PROGRAM RTC 
VAR
	FB_LocalSystemTime_0	: FB_LocalSystemTime;
	TimeStamp		: TIMESTRUCT;
		
	TimeStamp_GMT		: TIMESTRUCT;
	
	FB_GetTimeZoneInformation_0 :FB_GetTimeZoneInformation;
	FB_SetTimeZoneInformation_0	:FB_SetTimeZoneInformation;
	ST_TimeZoneInformation:ST_TimeZoneInformation;

	
	Timer :ton;
	FlagGetTimeZone:BOOL;// :=TRUE;
	FlagSetTimeZone:BOOL;// :=TRUE;
	FlagInit	   :BOOL :=TRUE;	
	
	ErrorIDGetTimeZone:UDINT;
	ErrorIDSetTimeZone:UDINT;
	
	FB_TzSpecificLocalTimeToSystemTime:FB_TzSpecificLocalTimeToSystemTime;
//	amsid:T_AmsNetID :='192.168.101.2.1.1' ;
	amsid:T_AmsNetID ;
	
	//IISreset
	NT_StartProcess:NT_StartProcess;
	Flagiisreset:BOOL;
END_VAR

//Timer(IN:=FlagInit,PT:=T#5S,Q=>FlagGetTimeZone);

FB_LocalSystemTime_0(
	sNetID:= '' , 
	bEnable:= TRUE, 
	dwCycle:= , 
	dwOpt:= , 
	tTimeout:= , 
	bValid=> , 
	systemTime=> TimeStamp, 
	tzID=> );

IF FlagInit THEN
	FlagGetTimeZone:=TRUE;
	Flagiisreset:=TRUE;
	FlagInit:=FALSE;
	
END_IF	

	FB_GetTimeZoneInformation_0(bExecute := FlagGetTimeZone,sNetID:=PcTransmit.fbPcTransmit_0.RTC_amsid);
	IF FB_GetTimeZoneInformation_0.bError THEN
		FlagGetTimeZone:=FALSE;
		ErrorIDGetTimeZone:=FB_GetTimeZoneInformation_0.nErrID;
		FB_GetTimeZoneInformation_0(bExecute := FlagGetTimeZone);   		
	ELSIF FB_GetTimeZoneInformation_0.bBusy=FALSE AND FlagGetTimeZone THEN
		ST_TimeZoneInformation:=FB_GetTimeZoneInformation_0.tzInfo;	
		FlagGetTimeZone:=FALSE;
		FlagSetTimeZone:=TRUE;
		FB_GetTimeZoneInformation_0(bExecute := FlagGetTimeZone);	
	END_IF


	FB_SetTimeZoneInformation_0(bExecute:=FlagSetTimeZone, tzInfo:=ST_TimeZoneInformation);
	IF FB_SetTimeZoneInformation_0.bError THEN
		FlagSetTimeZone:=FALSE;
		ErrorIDSetTimeZone:=FB_SetTimeZoneInformation_0.nErrID;
		FB_SetTimeZoneInformation_0(bExecute := FlagSetTimeZone);   		
	ELSIF FB_SetTimeZoneInformation_0.bBusy=FALSE AND FlagSetTimeZone THEN
		FlagSetTimeZone:=FALSE;
		FB_SetTimeZoneInformation_0(bExecute := FlagGetTimeZone);	
	END_IF
	

FB_TzSpecificLocalTimeToSystemTime(in:=TimeStamp,tzInfo:=ST_TimeZoneInformation, out=>TimeStamp_GMT);

(*TEMPH:= DINT_TO_INT(ST_TimeZoneInformation.bias+ST_TimeZoneInformation.daylightBias)/60;

Temp_H:=(WORD_TO_INT(TimeStamp.wHour) +TEMPH)MOD(24) ;
IF Temp_H<0 THEN
	Temp_H:=Temp_H+24;
END_IF

TimeStamp_GMT :=TimeStamp;
TimeStamp_GMT.wHour:= INT_TO_WORD(Temp_H);*)

//IISRESET
IF Flagiisreset THEN
	NT_StartProcess.PATHSTR := 'C:\hp\iisreset.bat';
	NT_StartProcess.DIRNAME := 'C:\hp';
	NT_StartProcess.START :=TRUE;
	NT_StartProcess();
	IF NT_StartProcess.BUSY = FALSE THEN
		Flagiisreset:=FALSE;
		NT_StartProcess.START :=FALSE;
		NT_StartProcess();
	END_IF
END_IF

END_PROGRAM

(* stored: Version 1.1.0.1, ProductVersion 3.1.4024.3
   POU RTC: Id {50512f07-723a-0493-25f6-641df9e0db66}, SpecialFunc None *)
